FUNCTION F_AtPositionState : BOOL
    // Check if the motor is within the state bounds
VAR_INPUT
    stMotionStage: DUT_MotionStage;
    stPositionState: DUT_PositionState;
END_VAR
VAR
END_VAR

F_AtPositionState := FALSE;
// We can never be at invalid states. We are also not at a state if a move has been requested, we are instead transitioning.
IF stPositionState.bValid AND NOT stMotionStage.bExecute THEN
    IF stMotionStage.stAxisStatus.fActPosition < stPositionState.fPosition + ABS(stPositionState.fDelta) AND
       stMotionStage.stAxisStatus.fActPosition > stPositionState.fPosition - ABS(stPositionState.fDelta) THEN
       F_AtPositionState := TRUE;
    END_IF
END_IF

END_FUNCTION

(* stored: Version 1.1.0.1, ProductVersion 3.1.4022.18
   POU F_AtPositionState: Id {058abbc4-740d-4ed6-b83c-7fdc99dbdef5}, SpecialFunc None *)
